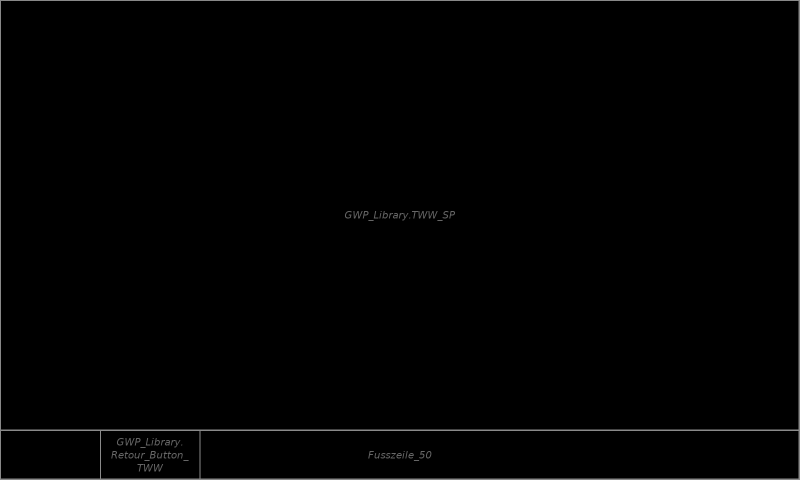
VISUALIZATION TWW_SP  // 800x480
    Frame (0,0 800x430)
        shows GWP_Library.TWW_SP(FB_TWW_SP := Main.TWW_SP_0, FB_Zirk_Pumpe := Main.Zirk_Pumpe_0, FB_Zusatzheizung := Main.Zusatzheizung_0, FB_KD := Main.KD_0)
    Group (0,430 800x50)
        Frame (0,0 800x50)
            shows Fusszeile_50()
        Frame (100,0 100x50)
            shows GWP_Library.Retour_Button_TWW()
END_VISUALIZATION

(* stored: Version 1.1.0.1, ProductVersion 3.1.4022.6
   Visu TWW_SP: Id {f81b9d4e-b1ca-4424-be75-82928e44433e} *)
